// TwinCAT 3 PLC project ElevatorControl
// ProgramVersion: 3.1.4024.0
// libraries:
//   Tc2_Standard, * (Beckhoff Automation GmbH)
//   Tc2_System, * (Beckhoff Automation GmbH)
//   Tc2_Utilities, * (Beckhoff Automation GmbH)
//   Tc3_Module, * (Beckhoff Automation GmbH)
// project tree:
//   DUTs/ AT_AlarmLog.TcDUT (not stored), AT_FloorCalls.TcDUT (not stored), E_AlarmSeverity.TcDUT (not stored), E_Direction.TcDUT (not stored), E_ElevatorState.TcDUT, E_TrafficMode.TcDUT (not stored), ST_AlarmEvent.TcDUT (not stored), ST_ElevatorStatus.TcDUT, ST_FloorCall.TcDUT, ST_PerformanceMetrics.TcDUT (not stored)
//   GVLs/ GVL_HMI.TcGVL, GVL_IO.TcGVL (not stored), GVL_Parameters.TcGVL (not stored)
//   / PlcTask.TcTTO
//   POUs/ FB_Elevator.TcPOU (not stored), FB_Safety.TcPOU, MAIN.TcPOU, FB_Dispatcher.TcPOU, PRG_Test_Elevator.TcPOU
// real-time tasks:
//   TASK PlcTask: cycle T#10ms, priority 20, ADS port 350
//   TASK PlcTask1: cycle T#10ms, priority 21, ADS port 351

CONFIGURATION ElevatorControl
    RESOURCE PLC ON TwinCAT3
        TASK PlcTask(INTERVAL := T#10ms, PRIORITY := 20);
        PROGRAM MAIN WITH PlcTask : MAIN;
    END_RESOURCE
END_CONFIGURATION

// ---- DUTs/E_ElevatorState.TcDUT
{attribute 'qualified_only'}
{attribute 'strict'}
TYPE E_ElevatorState :
(
	eIdle           := 0,   // Waiting for calls, doors closed
    eMovingUp       := 1,   // Traveling upward
    eMovingDown     := 2,   // Traveling downward
    eDoorsOpening   := 3,   // Door opening animation
    eDoorsOpen      := 4,   // Doors fully open, waiting for passengers
    eDoorsClosing   := 5,   // Door closing animation
    eEmergencyStop  := 6,   // Emergency stop button pressed
    eFireMode       := 7,   // Fire alarm — returning to ground
    eOverload       := 8,   // Too much weight detected
    eMaintenance    := 9    // Service mode (future feature)
);
END_TYPE

// ---- DUTs/ST_ElevatorStatus.TcDUT
TYPE ST_ElevatorStatus :
STRUCT
    iElevatorID     : INT;              // 1 = E1, 2 = E2
    iCurrentFloor   : INT;              // Which floor it's at (0-10)
    fPosition       : REAL;             // Smooth position 0.0-10.0 for animation
    eState          : E_ElevatorState;  // What it's doing right now
    eDirection      : E_Direction;      // Which way it's going
    bDoorsOpen      : BOOL;             // TRUE = doors are open
    fDoorOpenPercent: REAL;             // 0.0-100.0 for door animation width
    iNextTarget     : INT;              // Next floor it's going to (-1 = none)
    iQueueLength    : INT;              // How many calls pending
    bOverload       : BOOL;             // TRUE = too heavy
    bDoorObstruction: BOOL;             // TRUE = something blocking door
    fTravelDistance : REAL;             // Total meters traveled (maintenance metric)
    iTripCount      : DINT;             // Total completed trips
    tLastMaintenance: TIME;             // Time since last service
END_STRUCT
END_TYPE

// ---- DUTs/ST_FloorCall.TcDUT
TYPE ST_FloorCall :
STRUCT
    iFloor          : INT;          // Which floor (0 = Ground, 1-10)
    eDirection      : E_Direction;  // For hall buttons: Up or Down
    bIsCarCall      : BOOL;         // TRUE = pressed inside elevator, FALSE = hallway
    tTimestamp      : TIME;         // When the button was pressed
    iAssignedTo     : INT;          // 0 = not assigned yet, 1 = E1, 2 = E2
    bIsActive       : BOOL;         // TRUE = still waiting, FALSE = completed
    tWaitTime       : TIME;         // How long the person has been waiting
END_STRUCT
END_TYPE

// ---- GVLs/GVL_HMI.TcGVL
{attribute 'qualified_only'}
// ============================================
// GVL_HMI — Variables Exposed to HMI
// ============================================

VAR_GLOBAL
    // Elevator status — what the HMI displays
    g_stE1Status        : ST_ElevatorStatus;    // Everything about E1
    g_stE2Status        : ST_ElevatorStatus;    // Everything about E2
    
    // System metrics
    g_stMetrics         : ST_PerformanceMetrics;
    
    // Alarm history
    g_astAlarmLog       : AT_AlarmLog;
    g_iAlarmCount       : INT := 0;
    
    // Call queue display
    g_astCallQueue      : AT_FloorCalls;
    g_iQueueCount       : INT := 0;
    
    // System status text
    g_bSystemReady      		: BOOL := FALSE;
    g_sSystemStatus     		: STRING(40) := 'Initializing';
    g_bAlarmActive      		: BOOL := FALSE;
    g_sAlarmMessage     		: STRING(120) := '';
	g_bHMI_ResetAlarmEnabled 	: BOOL := FALSE;
    
    // ------------------------------------------------------------------------
    // HMI TO PLC — Commands from operator
    // ------------------------------------------------------------------------
    g_bHMI_EmergencyStop    : BOOL := FALSE;    // Pressed = stop everything
    g_bHMI_ResetEmergency   : BOOL := FALSE;    // Pressed = clear emergency
    g_bHMI_FireMode         : BOOL := FALSE;    // Pressed = activate fire mode
    g_bHMI_ResetFireMode    : BOOL := FALSE;    // Pressed = clear fire mode
    g_eHMI_TrafficMode      : E_TrafficMode := E_TrafficMode.eOffPeak;
    g_bHMI_ClearAllCalls    : BOOL := FALSE;    // Pressed = empty all queues
	g_bHMI_ResetAlarm 		: BOOL := FALSE;	// Pressed = reset active alarms
    
    // ------------------------------------------------------------------------
    // HMI TO PLC — Floor calls from HMI buttons
    // ------------------------------------------------------------------------
    // Hall calls
    g_bHMI_Call_G_Up        : BOOL := FALSE;
    g_bHMI_Call_1_Up        : BOOL := FALSE;
    g_bHMI_Call_1_Down      : BOOL := FALSE;
    g_bHMI_Call_2_Up        : BOOL := FALSE;
    g_bHMI_Call_2_Down      : BOOL := FALSE;
    g_bHMI_Call_3_Up        : BOOL := FALSE;
    g_bHMI_Call_3_Down      : BOOL := FALSE;
    g_bHMI_Call_4_Up        : BOOL := FALSE;
    g_bHMI_Call_4_Down      : BOOL := FALSE;
    g_bHMI_Call_5_Up        : BOOL := FALSE;
    g_bHMI_Call_5_Down      : BOOL := FALSE;
    g_bHMI_Call_6_Up        : BOOL := FALSE;
    g_bHMI_Call_6_Down      : BOOL := FALSE;
    g_bHMI_Call_7_Up        : BOOL := FALSE;
    g_bHMI_Call_7_Down      : BOOL := FALSE;
    g_bHMI_Call_8_Up        : BOOL := FALSE;
    g_bHMI_Call_8_Down      : BOOL := FALSE;
    g_bHMI_Call_9_Up        : BOOL := FALSE;
    g_bHMI_Call_9_Down      : BOOL := FALSE;
    g_bHMI_Call_10_Down     : BOOL := FALSE;
    
    // Car calls — Elevator 1
    g_bHMI_E1_Car_G         : BOOL := FALSE;
    g_bHMI_E1_Car_1         : BOOL := FALSE;
    g_bHMI_E1_Car_2         : BOOL := FALSE;
    g_bHMI_E1_Car_3         : BOOL := FALSE;
    g_bHMI_E1_Car_4         : BOOL := FALSE;
    g_bHMI_E1_Car_5         : BOOL := FALSE;
    g_bHMI_E1_Car_6         : BOOL := FALSE;
    g_bHMI_E1_Car_7         : BOOL := FALSE;
    g_bHMI_E1_Car_8         : BOOL := FALSE;
    g_bHMI_E1_Car_9         : BOOL := FALSE;
    g_bHMI_E1_Car_10        : BOOL := FALSE;
    
    // Car calls — Elevator 2
    g_bHMI_E2_Car_G         : BOOL := FALSE;
    g_bHMI_E2_Car_1         : BOOL := FALSE;
    g_bHMI_E2_Car_2         : BOOL := FALSE;
    g_bHMI_E2_Car_3         : BOOL := FALSE;
    g_bHMI_E2_Car_4         : BOOL := FALSE;
    g_bHMI_E2_Car_5         : BOOL := FALSE;
    g_bHMI_E2_Car_6         : BOOL := FALSE;
    g_bHMI_E2_Car_7         : BOOL := FALSE;
    g_bHMI_E2_Car_8         : BOOL := FALSE;
    g_bHMI_E2_Car_9         : BOOL := FALSE;
    g_bHMI_E2_Car_10        : BOOL := FALSE;
    
END_VAR

// ---- POUs/MAIN.TcPOU
PROGRAM MAIN

// ============================================================================
// ELEVATOR INSTANCES
// ============================================================================
VAR
    E1              : FB_Elevator;
    E2              : FB_Elevator;
	
	 prgTestElevator : PRG_Test_Elevator;

END_VAR

// ============================================================================
// GROUP CONTROL
// ============================================================================
VAR
    Dispatcher      : FB_Dispatcher;
END_VAR

// ============================================================================
// SAFETY SYSTEM
// ============================================================================
VAR
    Safety          : FB_Safety;
END_VAR

// ============================================================================
// SIMULATION INPUTS (Delete these when connecting real hardware)
// ============================================================================
VAR
    // Hall call simulation
    bSimHall_G_Up       : BOOL := FALSE;
    bSimHall_1_Up       : BOOL := FALSE;
    bSimHall_1_Down     : BOOL := FALSE;
    bSimHall_2_Up       : BOOL := FALSE;
    bSimHall_2_Down     : BOOL := FALSE;
    bSimHall_3_Up       : BOOL := FALSE;
    bSimHall_3_Down     : BOOL := FALSE;
    bSimHall_4_Up       : BOOL := FALSE;
    bSimHall_4_Down     : BOOL := FALSE;
    bSimHall_5_Up       : BOOL := FALSE;
    bSimHall_5_Down     : BOOL := FALSE;
    bSimHall_6_Up       : BOOL := FALSE;
    bSimHall_6_Down     : BOOL := FALSE;
    bSimHall_7_Up       : BOOL := FALSE;
    bSimHall_7_Down     : BOOL := FALSE;
    bSimHall_8_Up       : BOOL := FALSE;
    bSimHall_8_Down     : BOOL := FALSE;
    bSimHall_9_Up       : BOOL := FALSE;
    bSimHall_9_Down     : BOOL := FALSE;
    bSimHall_10_Down    : BOOL := FALSE;
    
    // Car call simulation — E1
    bSimE1_Car_G        : BOOL := FALSE;
    bSimE1_Car_1        : BOOL := FALSE;
    bSimE1_Car_2        : BOOL := FALSE;
    bSimE1_Car_3        : BOOL := FALSE;
    bSimE1_Car_4        : BOOL := FALSE;
    bSimE1_Car_5        : BOOL := FALSE;
    bSimE1_Car_6        : BOOL := FALSE;
    bSimE1_Car_7        : BOOL := FALSE;
    bSimE1_Car_8        : BOOL := FALSE;
    bSimE1_Car_9        : BOOL := FALSE;
    bSimE1_Car_10       : BOOL := FALSE;
    
    // Car call simulation — E2
    bSimE2_Car_G        : BOOL := FALSE;
    bSimE2_Car_1        : BOOL := FALSE;
    bSimE2_Car_2        : BOOL := FALSE;
    bSimE2_Car_3        : BOOL := FALSE;
    bSimE2_Car_4        : BOOL := FALSE;
    bSimE2_Car_5        : BOOL := FALSE;
    bSimE2_Car_6        : BOOL := FALSE;
    bSimE2_Car_7        : BOOL := FALSE;
    bSimE2_Car_8        : BOOL := FALSE;
    bSimE2_Car_9        : BOOL := FALSE;
    bSimE2_Car_10       : BOOL := FALSE;
    
    // Safety simulation
    bSimE1_DoorSensor   : BOOL := FALSE;
    bSimE1_WeightSensor : BOOL := FALSE;
    bSimE1_EmergencyBtn : BOOL := FALSE;
    bSimE2_DoorSensor   : BOOL := FALSE;
    bSimE2_WeightSensor : BOOL := FALSE;
    bSimE2_EmergencyBtn : BOOL := FALSE;
    bSimFireAlarm       : BOOL := FALSE;
    bSimPowerFault      : BOOL := FALSE;
    
    // HMI command simulation
    bSimHMI_EmergencyStop   : BOOL := FALSE;
    bSimHMI_ResetEmergency  : BOOL := FALSE;
    bSimHMI_FireMode        : BOOL := FALSE;
    bSimHMI_ResetFireMode   : BOOL := FALSE;
    bSimHMI_ClearAllCalls   : BOOL := FALSE;
END_VAR

// ============================================================================
// INTERNAL STATE TRACKING
// ============================================================================
VAR
    _bInitialized       : BOOL := FALSE;
    _bPrevClearCalls    : BOOL := FALSE;
	 bSystemEnable 		: BOOL := TRUE;
END_VAR

prgTestElevator();

// ======================================================================
// ONE-TIME INITIALIZATION
// ======================================================================
IF NOT _bInitialized THEN
    
    // Connect dispatcher references to elevator instances
    Dispatcher.refE1 REF= E1;
    Dispatcher.refE2 REF= E2;
    
    // Connect safety references to elevator instances
    Safety.refE1 REF= E1;
    Safety.refE2 REF= E2;
    
    _bInitialized := TRUE;
    
END_IF;

// ======================================================================
// SIMULATION: COPY SIM INPUTS TO PHYSICAL I/O ADDRESSES
// ======================================================================
// DELETE THIS ENTIRE SECTION WHEN CONNECTING REAL HARDWARE
// ----------------------------------------------------------------------

// Hall calls
GVL_IO.diHall_G_Up         := bSimHall_G_Up;
GVL_IO.diHall_1_Up         := bSimHall_1_Up;
GVL_IO.diHall_1_Down       := bSimHall_1_Down;
GVL_IO.diHall_2_Up         := bSimHall_2_Up;
GVL_IO.diHall_2_Down       := bSimHall_2_Down;
GVL_IO.diHall_3_Up         := bSimHall_3_Up;
GVL_IO.diHall_3_Down       := bSimHall_3_Down;
GVL_IO.diHall_4_Up         := bSimHall_4_Up;
GVL_IO.diHall_4_Down       := bSimHall_4_Down;
GVL_IO.diHall_5_Up         := bSimHall_5_Up;
GVL_IO.diHall_5_Down       := bSimHall_5_Down;
GVL_IO.diHall_6_Up         := bSimHall_6_Up;
GVL_IO.diHall_6_Down       := bSimHall_6_Down;
GVL_IO.diHall_7_Up         := bSimHall_7_Up;
GVL_IO.diHall_7_Down       := bSimHall_7_Down;
GVL_IO.diHall_8_Up         := bSimHall_8_Up;
GVL_IO.diHall_8_Down       := bSimHall_8_Down;
GVL_IO.diHall_9_Up         := bSimHall_9_Up;
GVL_IO.diHall_9_Down       := bSimHall_9_Down;
GVL_IO.diHall_10_Down      := bSimHall_10_Down;

// Car calls E1
GVL_IO.diE1_Car_G          := bSimE1_Car_G;
GVL_IO.diE1_Car_1          := bSimE1_Car_1;
GVL_IO.diE1_Car_2          := bSimE1_Car_2;
GVL_IO.diE1_Car_3          := bSimE1_Car_3;
GVL_IO.diE1_Car_4          := bSimE1_Car_4;
GVL_IO.diE1_Car_5          := bSimE1_Car_5;
GVL_IO.diE1_Car_6          := bSimE1_Car_6;
GVL_IO.diE1_Car_7          := bSimE1_Car_7;
GVL_IO.diE1_Car_8          := bSimE1_Car_8;
GVL_IO.diE1_Car_9          := bSimE1_Car_9;
GVL_IO.diE1_Car_10         := bSimE1_Car_10;

// Car calls E2
GVL_IO.diE2_Car_G          := bSimE2_Car_G;
GVL_IO.diE2_Car_1          := bSimE2_Car_1;
GVL_IO.diE2_Car_2          := bSimE2_Car_2;
GVL_IO.diE2_Car_3          := bSimE2_Car_3;
GVL_IO.diE2_Car_4          := bSimE2_Car_4;
GVL_IO.diE2_Car_5          := bSimE2_Car_5;
GVL_IO.diE2_Car_6          := bSimE2_Car_6;
GVL_IO.diE2_Car_7          := bSimE2_Car_7;
GVL_IO.diE2_Car_8          := bSimE2_Car_8;
GVL_IO.diE2_Car_9          := bSimE2_Car_9;
GVL_IO.diE2_Car_10         := bSimE2_Car_10;

// Safety sensors
GVL_IO.diE1_DoorSensor     := bSimE1_DoorSensor;
GVL_IO.diE1_WeightSensor   := bSimE1_WeightSensor;
GVL_IO.diE1_EmergencyBtn   := bSimE1_EmergencyBtn;
GVL_IO.diE2_DoorSensor     := bSimE2_DoorSensor;
GVL_IO.diE2_WeightSensor   := bSimE2_WeightSensor;
GVL_IO.diE2_EmergencyBtn   := bSimE2_EmergencyBtn;
GVL_IO.diFireAlarm         := bSimFireAlarm;
GVL_IO.diPowerFault        := bSimPowerFault;

// HMI commands
GVL_HMI.g_bHMI_EmergencyStop    := bSimHMI_EmergencyStop;
GVL_HMI.g_bHMI_ResetEmergency   := bSimHMI_ResetEmergency;
GVL_HMI.g_bHMI_FireMode         := bSimHMI_FireMode;
GVL_HMI.g_bHMI_ResetFireMode    := bSimHMI_ResetFireMode;
GVL_HMI.g_bHMI_ClearAllCalls    := bSimHMI_ClearAllCalls;

// ======================================================================
// MAP PHYSICAL I/O TO ELEVATOR INPUTS
// ======================================================================

// Elevator 1 inputs
E1.bEnable          := bSystemEnable AND Safety.bE1Enable;
E1.bEmergencyStop   := GVL_IO.diE1_EmergencyBtn OR GVL_HMI.g_bHMI_EmergencyStop;
E1.bFireMode        := GVL_IO.diFireAlarm OR GVL_HMI.g_bHMI_FireMode;
E1.bDoorObstruction := GVL_IO.diE1_DoorSensor;
E1.bOverload        := GVL_IO.diE1_WeightSensor;

// Elevator 2 inputs
E2.bEnable          := bSystemEnable AND Safety.bE2Enable;
E2.bEmergencyStop   := GVL_IO.diE2_EmergencyBtn OR GVL_HMI.g_bHMI_EmergencyStop;
E2.bFireMode        := GVL_IO.diFireAlarm OR GVL_HMI.g_bHMI_FireMode;
E2.bDoorObstruction := GVL_IO.diE2_DoorSensor;
E2.bOverload        := GVL_IO.diE2_WeightSensor;

// ======================================================================
// MAP PHYSICAL I/O TO SAFETY INPUTS
// ======================================================================
Safety.bE1DoorSensor    := GVL_IO.diE1_DoorSensor;
Safety.bE2DoorSensor    := GVL_IO.diE2_DoorSensor;
Safety.bE1WeightSensor  := GVL_IO.diE1_WeightSensor;
Safety.bE2WeightSensor  := GVL_IO.diE2_WeightSensor;
Safety.bE1EmergencyBtn  := GVL_IO.diE1_EmergencyBtn;
Safety.bE2EmergencyBtn  := GVL_IO.diE2_EmergencyBtn;
Safety.bFireAlarm       := GVL_IO.diFireAlarm;
Safety.bPowerFault      := GVL_IO.diPowerFault;

// ======================================================================
// PROCESS HALL CALLS → DISPATCHER
// ======================================================================
IF GVL_IO.diHall_G_Up      THEN Dispatcher.AddCall(0, E_Direction.eUp, FALSE, 0); END_IF;
IF GVL_IO.diHall_1_Up      THEN Dispatcher.AddCall(1, E_Direction.eUp, FALSE, 0); END_IF;
IF GVL_IO.diHall_1_Down    THEN Dispatcher.AddCall(1, E_Direction.eDown, FALSE, 0); END_IF;
IF GVL_IO.diHall_2_Up      THEN Dispatcher.AddCall(2, E_Direction.eUp, FALSE, 0); END_IF;
IF GVL_IO.diHall_2_Down    THEN Dispatcher.AddCall(2, E_Direction.eDown, FALSE, 0); END_IF;
IF GVL_IO.diHall_3_Up      THEN Dispatcher.AddCall(3, E_Direction.eUp, FALSE, 0); END_IF;
IF GVL_IO.diHall_3_Down    THEN Dispatcher.AddCall(3, E_Direction.eDown, FALSE, 0); END_IF;
IF GVL_IO.diHall_4_Up      THEN Dispatcher.AddCall(4, E_Direction.eUp, FALSE, 0); END_IF;
IF GVL_IO.diHall_4_Down    THEN Dispatcher.AddCall(4, E_Direction.eDown, FALSE, 0); END_IF;
IF GVL_IO.diHall_5_Up      THEN Dispatcher.AddCall(5, E_Direction.eUp, FALSE, 0); END_IF;
IF GVL_IO.diHall_5_Down    THEN Dispatcher.AddCall(5, E_Direction.eDown, FALSE, 0); END_IF;
IF GVL_IO.diHall_6_Up      THEN Dispatcher.AddCall(6, E_Direction.eUp, FALSE, 0); END_IF;
IF GVL_IO.diHall_6_Down    THEN Dispatcher.AddCall(6, E_Direction.eDown, FALSE, 0); END_IF;
IF GVL_IO.diHall_7_Up      THEN Dispatcher.AddCall(7, E_Direction.eUp, FALSE, 0); END_IF;
IF GVL_IO.diHall_7_Down    THEN Dispatcher.AddCall(7, E_Direction.eDown, FALSE, 0); END_IF;
IF GVL_IO.diHall_8_Up      THEN Dispatcher.AddCall(8, E_Direction.eUp, FALSE, 0); END_IF;
IF GVL_IO.diHall_8_Down    THEN Dispatcher.AddCall(8, E_Direction.eDown, FALSE, 0); END_IF;
IF GVL_IO.diHall_9_Up      THEN Dispatcher.AddCall(9, E_Direction.eUp, FALSE, 0); END_IF;
IF GVL_IO.diHall_9_Down    THEN Dispatcher.AddCall(9, E_Direction.eDown, FALSE, 0); END_IF;
IF GVL_IO.diHall_10_Down   THEN Dispatcher.AddCall(10, E_Direction.eDown, FALSE, 0); END_IF;

// ======================================================================
// PROCESS CAR CALLS → DIRECT TO ELEVATOR
// ======================================================================
IF GVL_IO.diE1_Car_G   THEN E1.CallFloor(0); END_IF;
IF GVL_IO.diE1_Car_1   THEN E1.CallFloor(1); END_IF;
IF GVL_IO.diE1_Car_2   THEN E1.CallFloor(2); END_IF;
IF GVL_IO.diE1_Car_3   THEN E1.CallFloor(3); END_IF;
IF GVL_IO.diE1_Car_4   THEN E1.CallFloor(4); END_IF;
IF GVL_IO.diE1_Car_5   THEN E1.CallFloor(5); END_IF;
IF GVL_IO.diE1_Car_6   THEN E1.CallFloor(6); END_IF;
IF GVL_IO.diE1_Car_7   THEN E1.CallFloor(7); END_IF;
IF GVL_IO.diE1_Car_8   THEN E1.CallFloor(8); END_IF;
IF GVL_IO.diE1_Car_9   THEN E1.CallFloor(9); END_IF;
IF GVL_IO.diE1_Car_10  THEN E1.CallFloor(10); END_IF;

IF GVL_IO.diE2_Car_G   THEN E2.CallFloor(0); END_IF;
IF GVL_IO.diE2_Car_1   THEN E2.CallFloor(1); END_IF;
IF GVL_IO.diE2_Car_2   THEN E2.CallFloor(2); END_IF;
IF GVL_IO.diE2_Car_3   THEN E2.CallFloor(3); END_IF;
IF GVL_IO.diE2_Car_4   THEN E2.CallFloor(4); END_IF;
IF GVL_IO.diE2_Car_5   THEN E2.CallFloor(5); END_IF;
IF GVL_IO.diE2_Car_6   THEN E2.CallFloor(6); END_IF;
IF GVL_IO.diE2_Car_7   THEN E2.CallFloor(7); END_IF;
IF GVL_IO.diE2_Car_8   THEN E2.CallFloor(8); END_IF;
IF GVL_IO.diE2_Car_9   THEN E2.CallFloor(9); END_IF;
IF GVL_IO.diE2_Car_10  THEN E2.CallFloor(10); END_IF;

// ======================================================================
// HMI CAR CALLS
// ======================================================================
IF GVL_HMI.g_bHMI_E1_Car_G THEN E1.CallFloor(0); GVL_HMI.g_bHMI_E1_Car_G := FALSE; END_IF;
IF GVL_HMI.g_bHMI_E1_Car_1 THEN E1.CallFloor(1); GVL_HMI.g_bHMI_E1_Car_1 := FALSE; END_IF;
IF GVL_HMI.g_bHMI_E1_Car_2 THEN E1.CallFloor(2); GVL_HMI.g_bHMI_E1_Car_2 := FALSE; END_IF;
IF GVL_HMI.g_bHMI_E1_Car_3 THEN E1.CallFloor(3); GVL_HMI.g_bHMI_E1_Car_3 := FALSE; END_IF;
IF GVL_HMI.g_bHMI_E1_Car_4 THEN E1.CallFloor(4); GVL_HMI.g_bHMI_E1_Car_4 := FALSE; END_IF;
IF GVL_HMI.g_bHMI_E1_Car_5 THEN E1.CallFloor(5); GVL_HMI.g_bHMI_E1_Car_5 := FALSE; END_IF;
IF GVL_HMI.g_bHMI_E1_Car_6 THEN E1.CallFloor(6); GVL_HMI.g_bHMI_E1_Car_6 := FALSE; END_IF;
IF GVL_HMI.g_bHMI_E1_Car_7 THEN E1.CallFloor(7); GVL_HMI.g_bHMI_E1_Car_7 := FALSE; END_IF;
IF GVL_HMI.g_bHMI_E1_Car_8 THEN E1.CallFloor(8); GVL_HMI.g_bHMI_E1_Car_8 := FALSE; END_IF;
IF GVL_HMI.g_bHMI_E1_Car_9 THEN E1.CallFloor(9); GVL_HMI.g_bHMI_E1_Car_9 := FALSE; END_IF;
IF GVL_HMI.g_bHMI_E1_Car_10 THEN E1.CallFloor(10); GVL_HMI.g_bHMI_E1_Car_10 := FALSE; END_IF;

IF GVL_HMI.g_bHMI_E2_Car_G THEN E2.CallFloor(0); GVL_HMI.g_bHMI_E2_Car_G := FALSE; END_IF;
IF GVL_HMI.g_bHMI_E2_Car_1 THEN E2.CallFloor(1); GVL_HMI.g_bHMI_E2_Car_1 := FALSE; END_IF;
IF GVL_HMI.g_bHMI_E2_Car_2 THEN E2.CallFloor(2); GVL_HMI.g_bHMI_E2_Car_2 := FALSE; END_IF;
IF GVL_HMI.g_bHMI_E2_Car_3 THEN E2.CallFloor(3); GVL_HMI.g_bHMI_E2_Car_3 := FALSE; END_IF;
IF GVL_HMI.g_bHMI_E2_Car_4 THEN E2.CallFloor(4); GVL_HMI.g_bHMI_E2_Car_4 := FALSE; END_IF;
IF GVL_HMI.g_bHMI_E2_Car_5 THEN E2.CallFloor(5); GVL_HMI.g_bHMI_E2_Car_5 := FALSE; END_IF;
IF GVL_HMI.g_bHMI_E2_Car_6 THEN E2.CallFloor(6); GVL_HMI.g_bHMI_E2_Car_6 := FALSE; END_IF;
IF GVL_HMI.g_bHMI_E2_Car_7 THEN E2.CallFloor(7); GVL_HMI.g_bHMI_E2_Car_7 := FALSE; END_IF;
IF GVL_HMI.g_bHMI_E2_Car_8 THEN E2.CallFloor(8); GVL_HMI.g_bHMI_E2_Car_8 := FALSE; END_IF;
IF GVL_HMI.g_bHMI_E2_Car_9 THEN E2.CallFloor(9); GVL_HMI.g_bHMI_E2_Car_9 := FALSE; END_IF;
IF GVL_HMI.g_bHMI_E2_Car_10 THEN E2.CallFloor(10); GVL_HMI.g_bHMI_E2_Car_10 := FALSE; END_IF;

// ======================================================================
// HMI HALL CALLS
// ======================================================================
IF GVL_HMI.g_bHMI_Call_G_Up THEN Dispatcher.AddCall(0, E_Direction.eUp, FALSE, 0); GVL_HMI.g_bHMI_Call_G_Up := FALSE; END_IF;
IF GVL_HMI.g_bHMI_Call_1_Up THEN Dispatcher.AddCall(1, E_Direction.eUp, FALSE, 0); GVL_HMI.g_bHMI_Call_1_Up := FALSE; END_IF;
IF GVL_HMI.g_bHMI_Call_1_Down THEN Dispatcher.AddCall(1, E_Direction.eDown, FALSE, 0); GVL_HMI.g_bHMI_Call_1_Down := FALSE; END_IF;
IF GVL_HMI.g_bHMI_Call_2_Up THEN Dispatcher.AddCall(2, E_Direction.eUp, FALSE, 0); GVL_HMI.g_bHMI_Call_2_Up := FALSE; END_IF;
IF GVL_HMI.g_bHMI_Call_2_Down THEN Dispatcher.AddCall(2, E_Direction.eDown, FALSE, 0); GVL_HMI.g_bHMI_Call_2_Down := FALSE; END_IF;
IF GVL_HMI.g_bHMI_Call_3_Up THEN Dispatcher.AddCall(3, E_Direction.eUp, FALSE, 0); GVL_HMI.g_bHMI_Call_3_Up := FALSE; END_IF;
IF GVL_HMI.g_bHMI_Call_3_Down THEN Dispatcher.AddCall(3, E_Direction.eDown, FALSE, 0); GVL_HMI.g_bHMI_Call_3_Down := FALSE; END_IF;
IF GVL_HMI.g_bHMI_Call_4_Up THEN Dispatcher.AddCall(4, E_Direction.eUp, FALSE, 0); GVL_HMI.g_bHMI_Call_4_Up := FALSE; END_IF;
IF GVL_HMI.g_bHMI_Call_4_Down THEN Dispatcher.AddCall(4, E_Direction.eDown, FALSE, 0); GVL_HMI.g_bHMI_Call_4_Down := FALSE; END_IF;
IF GVL_HMI.g_bHMI_Call_5_Up THEN Dispatcher.AddCall(5, E_Direction.eUp, FALSE, 0); GVL_HMI.g_bHMI_Call_5_Up := FALSE; END_IF;
IF GVL_HMI.g_bHMI_Call_5_Down THEN Dispatcher.AddCall(5, E_Direction.eDown, FALSE, 0); GVL_HMI.g_bHMI_Call_5_Down := FALSE; END_IF;
IF GVL_HMI.g_bHMI_Call_6_Up THEN Dispatcher.AddCall(6, E_Direction.eUp, FALSE, 0); GVL_HMI.g_bHMI_Call_6_Up := FALSE; END_IF;
IF GVL_HMI.g_bHMI_Call_6_Down THEN Dispatcher.AddCall(6, E_Direction.eDown, FALSE, 0); GVL_HMI.g_bHMI_Call_6_Down := FALSE; END_IF;
IF GVL_HMI.g_bHMI_Call_7_Up THEN Dispatcher.AddCall(7, E_Direction.eUp, FALSE, 0); GVL_HMI.g_bHMI_Call_7_Up := FALSE; END_IF;
IF GVL_HMI.g_bHMI_Call_7_Down THEN Dispatcher.AddCall(7, E_Direction.eDown, FALSE, 0); GVL_HMI.g_bHMI_Call_7_Down := FALSE; END_IF;
IF GVL_HMI.g_bHMI_Call_8_Up THEN Dispatcher.AddCall(8, E_Direction.eUp, FALSE, 0); GVL_HMI.g_bHMI_Call_8_Up := FALSE; END_IF;
IF GVL_HMI.g_bHMI_Call_8_Down THEN Dispatcher.AddCall(8, E_Direction.eDown, FALSE, 0); GVL_HMI.g_bHMI_Call_8_Down := FALSE; END_IF;
IF GVL_HMI.g_bHMI_Call_9_Up THEN Dispatcher.AddCall(9, E_Direction.eUp, FALSE, 0); GVL_HMI.g_bHMI_Call_9_Up := FALSE; END_IF;
IF GVL_HMI.g_bHMI_Call_9_Down THEN Dispatcher.AddCall(9, E_Direction.eDown, FALSE, 0); GVL_HMI.g_bHMI_Call_9_Down := FALSE; END_IF;
IF GVL_HMI.g_bHMI_Call_10_Down THEN Dispatcher.AddCall(10, E_Direction.eDown, FALSE, 0); GVL_HMI.g_bHMI_Call_10_Down := FALSE; END_IF;

// ======================================================================
// RESET ACTIVE ALARM (HMI command)
// ======================================================================
IF GVL_HMI.g_bHMI_ResetAlarm THEN
    IF Safety.ResetSystemAlarm() THEN
        GVL_HMI.g_bHMI_ResetAlarm := FALSE;
    END_IF
END_IF;

// ======================================================================
// CLEAR ALL CALLS
// ======================================================================
IF GVL_HMI.g_bHMI_ClearAllCalls AND NOT _bPrevClearCalls THEN
    Dispatcher.ClearAllCalls();
    E1.ClearCall(0); E1.ClearCall(1); E1.ClearCall(2); E1.ClearCall(3);
    E1.ClearCall(4); E1.ClearCall(5); E1.ClearCall(6); E1.ClearCall(7);
    E1.ClearCall(8); E1.ClearCall(9); E1.ClearCall(10);
    E2.ClearCall(0); E2.ClearCall(1); E2.ClearCall(2); E2.ClearCall(3);
    E2.ClearCall(4); E2.ClearCall(5); E2.ClearCall(6); E2.ClearCall(7);
    E2.ClearCall(8); E2.ClearCall(9); E2.ClearCall(10);
END_IF;

_bPrevClearCalls := GVL_HMI.g_bHMI_ClearAllCalls;

// ======================================================================
// CYCLIC EXECUTION — CALL ALL FBs EVERY SCAN
// ======================================================================

// Run elevators
E1();
E2();

// Run dispatcher
Dispatcher.ProcessQueue();
Dispatcher.eTrafficMode := GVL_HMI.g_eHMI_TrafficMode;

// Run safety
Safety();

// ======================================================================
// UPDATE HMI OUTPUT DATA
// ======================================================================
GVL_HMI.g_stE1Status := E1.GetStatus();
GVL_HMI.g_stE2Status := E2.GetStatus();
GVL_HMI.g_stMetrics := Dispatcher.stMetrics;
GVL_HMI.g_astAlarmLog := Safety.GetAlarmLog();
GVL_HMI.g_bSystemReady := E1.bIsReady OR E2.bIsReady;
GVL_HMI.g_bAlarmActive := Safety.bSystemAlarm;
GVL_HMI.g_bHMI_ResetAlarmEnabled := Safety.bSystemAlarm;

IF Safety.bSystemAlarm THEN
    GVL_HMI.g_sAlarmMessage := Safety.sAlarmMessage;
ELSE
    GVL_HMI.g_sAlarmMessage := '';
END_IF;

// System status text
IF E1.eState = E_ElevatorState.eEmergencyStop OR 
   E2.eState = E_ElevatorState.eEmergencyStop THEN
    GVL_HMI.g_sSystemStatus := 'EMERGENCY STOP';
ELSIF E1.eState = E_ElevatorState.eFireMode OR 	
      E2.eState = E_ElevatorState.eFireMode THEN
    GVL_HMI.g_sSystemStatus := 'FIRE MODE ACTIVE';
ELSIF NOT bSystemEnable THEN
    GVL_HMI.g_sSystemStatus := 'SYSTEM DISABLED';
ELSE
    GVL_HMI.g_sSystemStatus := 'NORMAL OPERATION';
END_IF;

END_PROGRAM

// ---- POUs/PRG_Test_Elevator.TcPOU
FUNCTION_BLOCK PRG_Test_Elevator
VAR
    // Instance under test
    fbElev  : FB_Elevator;
    
    // Test control
    nStep       : INT := 0;
    bDone       : BOOL := FALSE;
    bPassed     : BOOL := FALSE;
    
    // Step timer
    tonWait     : TON;
    
    // Call tracking
    bCalledFloor3   : BOOL := FALSE;
    bCalledFloor1   : BOOL := FALSE;
END_VAR

// ============================================
// ELEVATOR UNIT TEST — Automatic Sequence
// ============================================

IF bDone THEN
    RETURN; // Test finished, keep results visible
END_IF;

CASE nStep OF

// --------------------------------------------
// STEP 0: Verify initial state
// --------------------------------------------
0:
    IF fbElev.eState = E_ElevatorState.eIdle AND 
       fbElev.iCurrentFloor = 0 AND
       fbElev.fDoorOpenPercent = 0.0 THEN
        nStep := 1;
    END_IF;

// --------------------------------------------
// STEP 1: Call elevator to floor 3
// --------------------------------------------
1:
    fbElev.bEnable := TRUE;
    IF NOT bCalledFloor3 THEN
        fbElev.CallFloor(3);
        bCalledFloor3 := TRUE;
    END_IF;
    
    // Should start moving up
    IF fbElev.eState = E_ElevatorState.eMovingUp THEN
        nStep := 2;
    END_IF;

// --------------------------------------------
// STEP 2: Wait until doors open at floor 3
// --------------------------------------------
2:
    IF fbElev.iCurrentFloor = 3 AND 
       fbElev.eState = E_ElevatorState.eDoorsOpen AND
       fbElev.fDoorOpenPercent >= 99.0 THEN
        nStep := 3;
        tonWait(IN := FALSE); // Reset timer
    END_IF;

// --------------------------------------------
// STEP 3: Wait for doors to close, return to idle
// --------------------------------------------
3:
    tonWait(IN := TRUE, PT := T#5S); // Give time for full cycle
    
    IF fbElev.eState = E_ElevatorState.eIdle AND tonWait.Q THEN
        nStep := 4;
        bCalledFloor1 := FALSE;
    END_IF;

// --------------------------------------------
// STEP 4: Call floor 1 (going down)
// --------------------------------------------
4:
    IF NOT bCalledFloor1 THEN
        fbElev.CallFloor(1);
        bCalledFloor1 := TRUE;
    END_IF;
    
    IF fbElev.eState = E_ElevatorState.eMovingDown THEN
        nStep := 5;
    END_IF;

// --------------------------------------------
// STEP 5: Arrive at floor 1, verify complete
// --------------------------------------------
5:
    IF fbElev.iCurrentFloor = 1 AND 
       fbElev.eState = E_ElevatorState.eIdle THEN
        bPassed := TRUE;
        bDone := TRUE;
    END_IF;

END_CASE;

// Call the function block every scan
//fbElev();

END_FUNCTION_BLOCK

// ---- POUs/FB_Dispatcher.TcPOU
FUNCTION_BLOCK FB_Dispatcher

// ============================================================================
// CONSTANTS
// ============================================================================
VAR CONSTANT
    cMAX_QUEUE_SIZE : INT := 50;
END_VAR

// ============================================================================
// INPUTS
// ============================================================================
VAR_INPUT
    // References to elevators (Composition pattern)
    refE1               : REFERENCE TO FB_Elevator;
    refE2               : REFERENCE TO FB_Elevator;
    
    // Traffic mode selection
    eTrafficMode        : E_TrafficMode := E_TrafficMode.eOffPeak;
    
    // System enable
    bEnable             : BOOL := TRUE;
END_VAR

// ============================================================================
// OUTPUTS
// ============================================================================
VAR_OUTPUT
    // Assignment tracking
    iAssignedToE1       : INT := 0;
    iAssignedToE2       : INT := 0;
    iUnassignedCalls    : INT := 0;
    
    // Performance metrics
    stMetrics           : ST_PerformanceMetrics;
END_VAR

// ============================================================================
// INTERNAL VARIABLES
// ============================================================================
VAR
    // Call queue
    _astCallQueue       : ARRAY[0..cMAX_QUEUE_SIZE] OF ST_FloorCall;
    _iQueueHead         : INT := 0;
    _iQueueTail         : INT := 0;
    _iQueueCount        : INT := 0;
    
    // Statistics
    _iTotalCalls        : DINT := 0;
    _fTotalWaitTime     : REAL := 0.0;
    _fMaxWaitTime       : REAL := 0.0;
    
    // Night mode
    _bNightModeActive   : BOOL := FALSE;
    _iActiveElevator    : INT := 1;
END_VAR

METHOD PUBLIC AddCall : BOOL
VAR_INPUT
    iFloor          : INT;
    eDirection      : E_Direction;
    bIsCarCall      : BOOL;
    iElevatorID     : INT;  // 0=hall call, 1=E1 car call, 2=E2 car call
END_VAR
IF _iQueueCount >= cMAX_QUEUE_SIZE THEN
    AddCall := FALSE;
    RETURN;
END_IF;

_astCallQueue[_iQueueTail].iFloor := iFloor;
_astCallQueue[_iQueueTail].eDirection := eDirection;
_astCallQueue[_iQueueTail].bIsCarCall := bIsCarCall;
_astCallQueue[_iQueueTail].tTimestamp := TIME();
_astCallQueue[_iQueueTail].iAssignedTo := 0;
_astCallQueue[_iQueueTail].bIsActive := TRUE;
_astCallQueue[_iQueueTail].tWaitTime := T#0S;

_iQueueTail := (_iQueueTail + 1) MOD (cMAX_QUEUE_SIZE + 1);
_iQueueCount := _iQueueCount + 1;
_iTotalCalls := _iTotalCalls + 1;

AddCall := TRUE;
END_METHOD

METHOD PRIVATE CalculateMetrics : BOOL
VAR
	fTotalDistance : REAL;
END_VAR
IF _iTotalCalls > 0 THEN
    stMetrics.fAvgResponseTime := _fTotalWaitTime / DINT_TO_REAL(_iTotalCalls);
ELSE
    stMetrics.fAvgResponseTime := 0.0;
END_IF;

stMetrics.fAvgWaitTime := stMetrics.fAvgResponseTime;
stMetrics.fMaxWaitTime := _fMaxWaitTime;

IF refE1.eState <> E_ElevatorState.eIdle AND 
   refE1.eState <> E_ElevatorState.eEmergencyStop THEN
    stMetrics.fUtilizationE1 := 85.0;
ELSE
    stMetrics.fUtilizationE1 := 15.0;
END_IF;

IF refE2.eState <> E_ElevatorState.eIdle AND 
   refE2.eState <> E_ElevatorState.eEmergencyStop THEN
    stMetrics.fUtilizationE2 := 85.0;
ELSE
    stMetrics.fUtilizationE2 := 15.0;
END_IF;

stMetrics.iCallsToday := _iTotalCalls;

fTotalDistance := refE1.fTravelDistance + refE2.fTravelDistance;
stMetrics.fEnergyEstimate := fTotalDistance * 0.15;

CalculateMetrics := TRUE;
END_METHOD

METHOD PUBLIC ClearAllCalls : BOOL
VAR
	i	: INT;
END_VAR
FOR i := 0 TO cMAX_QUEUE_SIZE DO
    _astCallQueue[i].bIsActive := FALSE;
END_FOR;

_iQueueCount := 0;
_iQueueHead := 0;
_iQueueTail := 0;

ClearAllCalls := TRUE;
END_METHOD

METHOD PUBLIC GetQueueStatus : AT_FloorCalls
VAR
	i : INT;
    j : INT := 0;
    aResult : AT_FloorCalls;
END_VAR
FOR i := 0 TO cMAX_QUEUE_SIZE DO
    IF _astCallQueue[i].bIsActive THEN
        aResult[j] := _astCallQueue[i];
        j := j + 1;
        IF j > cMAX_QUEUE_SIZE THEN
            EXIT;
        END_IF;
    END_IF;
END_FOR;

GetQueueStatus := aResult;
END_METHOD

METHOD ProcessQueue : BOOL
VAR
	i                   : INT;
    fScoreE1            : REAL;
    fScoreE2            : REAL;
    fDistanceE1         : REAL;
    fDistanceE2         : REAL;
    bE1CanServe         : BOOL;
    bE2CanServe         : BOOL;
    iE1Floor            : INT;
    iE2Floor            : INT;
    eE1Dir              : E_Direction;
    eE2Dir              : E_Direction;
    eE1State            : E_ElevatorState;
    eE2State            : E_ElevatorState;
END_VAR
IF NOT bEnable THEN
    ProcessQueue := FALSE;
    RETURN;
END_IF;


// 
iAssignedToE1 := 0;
iAssignedToE2 := 0;
iUnassignedCalls := 0;

// Get current elevator states
iE1Floor := refE1.iCurrentFloor;
iE2Floor := refE2.iCurrentFloor;
eE1Dir := refE1.eDirection;
eE2Dir := refE2.eDirection;
eE1State := refE1.eState;
eE2State := refE2.eState;

// Night mode handling
IF eTrafficMode = E_TrafficMode.eNightMode THEN
    IF NOT _bNightModeActive THEN
        _bNightModeActive := TRUE;
        IF _iActiveElevator = 1 THEN
            refE2.CallFloor(0);
        ELSE
            refE1.CallFloor(0);
        END_IF;
    END_IF;
ELSE
    _bNightModeActive := FALSE;
END_IF;

// Process each unassigned call
FOR i := 0 TO cMAX_QUEUE_SIZE DO
    IF _astCallQueue[i].bIsActive AND _astCallQueue[i].iAssignedTo = 0 THEN
        
        // Calculate distances
        fDistanceE1 := ABS(INT_TO_REAL(iE1Floor - _astCallQueue[i].iFloor));
        fDistanceE2 := ABS(INT_TO_REAL(iE2Floor - _astCallQueue[i].iFloor));
        
        // Direction compatibility
        bE1CanServe := (eE1Dir = E_Direction.eNone) OR 
                       (eE1Dir = _astCallQueue[i].eDirection) OR
                       _astCallQueue[i].bIsCarCall;
        bE2CanServe := (eE2Dir = E_Direction.eNone) OR 
                       (eE2Dir = _astCallQueue[i].eDirection) OR
                       _astCallQueue[i].bIsCarCall;
        
        // Base scores
        fScoreE1 := fDistanceE1;
        fScoreE2 := fDistanceE2;
        
        // Direction bonus
        IF bE1CanServe AND eE1Dir = _astCallQueue[i].eDirection THEN
            fScoreE1 := fScoreE1 * 0.6;
        END_IF;
        IF bE2CanServe AND eE2Dir = _astCallQueue[i].eDirection THEN
            fScoreE2 := fScoreE2 * 0.6;
        END_IF;
        
        // Traffic mode adjustments
        CASE eTrafficMode OF
            E_TrafficMode.eUpPeak:
                IF _astCallQueue[i].iFloor = 0 AND _astCallQueue[i].eDirection = E_Direction.eUp THEN
                    fScoreE1 := fScoreE1 * 0.7;
                END_IF;
                
            E_TrafficMode.eDownPeak:
                IF _astCallQueue[i].eDirection = E_Direction.eDown THEN
                    fScoreE2 := fScoreE2 * 0.7;
                END_IF;
                
            E_TrafficMode.eNightMode:
                IF _iActiveElevator = 1 THEN
                    fScoreE2 := 999.0;
                ELSE
                    fScoreE1 := 999.0;
                END_IF;
                
        END_CASE;
        
        // Availability check
        IF eE1State = E_ElevatorState.eEmergencyStop OR 
           eE1State = E_ElevatorState.eFireMode OR 
           eE1State = E_ElevatorState.eMaintenance THEN
            fScoreE1 := 999.0;
        END_IF;
        IF eE2State = E_ElevatorState.eEmergencyStop OR 
           eE2State = E_ElevatorState.eFireMode OR 
           eE2State = E_ElevatorState.eMaintenance THEN
            fScoreE2 := 999.0;
        END_IF;
        
        // Assign to best elevator
        IF fScoreE1 <= fScoreE2 THEN
            _astCallQueue[i].iAssignedTo := 1;
            refE1.CallFloor(_astCallQueue[i].iFloor);
            iAssignedToE1 := iAssignedToE1 + 1;
        ELSE
            _astCallQueue[i].iAssignedTo := 2;
            refE2.CallFloor(_astCallQueue[i].iFloor);
            iAssignedToE2 := iAssignedToE2 + 1;
        END_IF;
        
    END_IF;
END_FOR;

// Update completed calls and metrics
UpdateQueueStatus();
CalculateMetrics();

ProcessQueue := TRUE;
END_METHOD

METHOD PRIVATE UpdateQueueStatus : BOOL
VAR
	i : INT;
END_VAR
FOR i := 0 TO cMAX_QUEUE_SIZE DO
    IF _astCallQueue[i].bIsActive THEN
        
        // Update wait time
        _astCallQueue[i].tWaitTime := _astCallQueue[i].tWaitTime + TIME();
        
        // Check if call completed
        IF _astCallQueue[i].iAssignedTo = 1 THEN
            IF refE1.iCurrentFloor = _astCallQueue[i].iFloor AND 
               refE1.eState = E_ElevatorState.eDoorsOpen THEN
                _astCallQueue[i].bIsActive := FALSE;
                _iQueueCount := _iQueueCount - 1;
                
                _fTotalWaitTime := _fTotalWaitTime + TIME_TO_REAL(_astCallQueue[i].tWaitTime);
                IF TIME_TO_REAL(_astCallQueue[i].tWaitTime) > _fMaxWaitTime THEN
                    _fMaxWaitTime := TIME_TO_REAL(_astCallQueue[i].tWaitTime);
                END_IF;
            END_IF;
        ELSIF _astCallQueue[i].iAssignedTo = 2 THEN
            IF refE2.iCurrentFloor = _astCallQueue[i].iFloor AND 
               refE2.eState = E_ElevatorState.eDoorsOpen THEN
                _astCallQueue[i].bIsActive := FALSE;
                _iQueueCount := _iQueueCount - 1;
                
                _fTotalWaitTime := _fTotalWaitTime + TIME_TO_REAL(_astCallQueue[i].tWaitTime);
                IF TIME_TO_REAL(_astCallQueue[i].tWaitTime) > _fMaxWaitTime THEN
                    _fMaxWaitTime := TIME_TO_REAL(_astCallQueue[i].tWaitTime);
                END_IF;
            END_IF;
        END_IF;
        
    END_IF;
END_FOR;

UpdateQueueStatus := TRUE;
END_METHOD

END_FUNCTION_BLOCK

// ---- POUs/FB_Safety.TcPOU
FUNCTION_BLOCK FB_Safety

// ============================================================================
// CONSTANTS
// ============================================================================
VAR CONSTANT
    cMAX_ALARMS : INT := 99;
END_VAR

// ============================================================================
// INPUTS — Raw sensor signals
// ============================================================================
VAR_INPUT
    // Elevator references (to command them)
    refE1               : REFERENCE TO FB_Elevator;
    refE2               : REFERENCE TO FB_Elevator;
    
    // Door sensors (TRUE = obstruction detected)
    bE1DoorSensor       : BOOL := FALSE;
    bE2DoorSensor       : BOOL := FALSE;
    
    // Weight sensors (TRUE = overload)
    bE1WeightSensor     : BOOL := FALSE;
    bE2WeightSensor     : BOOL := FALSE;
    
    // Emergency stop buttons (TRUE = pressed)
    bE1EmergencyBtn     : BOOL := FALSE;
    bE2EmergencyBtn     : BOOL := FALSE;
    
    // Building safety
    bFireAlarm          : BOOL := FALSE;
    bFirefighterKey     : BOOL := FALSE;
    bPowerFault         : BOOL := FALSE;
    
    // Overspeed detectors
    bOverspeedE1        : BOOL := FALSE;
    bOverspeedE2        : BOOL := FALSE;
    
    // Door mechanism faults
    bDoorOpenFaultE1    : BOOL := FALSE;
    bDoorOpenFaultE2    : BOOL := FALSE;
END_VAR

// ============================================================================
// OUTPUTS — Safety decisions
// ============================================================================
VAR_OUTPUT
    bE1Enable           : BOOL := TRUE;
    bE2Enable           : BOOL := TRUE;
    bSystemAlarm        : BOOL := FALSE;
    sAlarmMessage       : STRING(120) := '';
    eAlarmSeverity      : E_AlarmSeverity := E_AlarmSeverity.eInfo;
    
    // Individual alarm flags
    bE1DoorObstruction  : BOOL := FALSE;
    bE2DoorObstruction  : BOOL := FALSE;
    bE1Overload         : BOOL := FALSE;
    bE2Overload         : BOOL := FALSE;
    bE1EmergencyActive  : BOOL := FALSE;
    bE2EmergencyActive  : BOOL := FALSE;
    bFireModeActive     : BOOL := FALSE;
END_VAR

// ============================================================================
// INTERNAL VARIABLES
// ============================================================================
VAR
    // Debounce timers
    _tonDoorObsE1       : TON;
    _tonDoorObsE2       : TON;
    _tonOverloadE1      : TON;
    _tonOverloadE2      : TON;
    _tonEmergencyE1     : TON;
    _tonEmergencyE2     : TON;
    _tonFireAlarm       : TON;
    _tonPowerFault      : TON;
    
    // Alarm history
    _astAlarmLog        : AT_AlarmLog;
    _iAlarmIndex        : INT := 0;
    _iNextEventID       : DINT := 1;
END_VAR

// ======================================================================
// DOOR OBSTRUCTION DETECTION
// ======================================================================
_tonDoorObsE1(IN := bE1DoorSensor, PT := T#200MS);
IF _tonDoorObsE1.Q THEN
    bE1DoorObstruction := TRUE;
    refE1.bDoorObstruction := TRUE;
    bSystemAlarm := TRUE;
    sAlarmMessage := 'E1 Door Obstruction Detected';
    eAlarmSeverity := E_AlarmSeverity.eWarning;
    AddAlarm(E_AlarmSeverity.eWarning, 1, 'E1 Door Obstruction', 'FB_Safety');
ELSE
    bE1DoorObstruction := FALSE;
    refE1.bDoorObstruction := FALSE;
END_IF;

_tonDoorObsE2(IN := bE2DoorSensor, PT := T#200MS);
IF _tonDoorObsE2.Q THEN
    bE2DoorObstruction := TRUE;
    refE2.bDoorObstruction := TRUE;
    bSystemAlarm := TRUE;
    sAlarmMessage := 'E2 Door Obstruction Detected';
    eAlarmSeverity := E_AlarmSeverity.eWarning;
    AddAlarm(E_AlarmSeverity.eWarning, 2, 'E2 Door Obstruction', 'FB_Safety');
ELSE
    bE2DoorObstruction := FALSE;
    refE2.bDoorObstruction := FALSE;
END_IF;

// ======================================================================
// OVERLOAD DETECTION
// ======================================================================
_tonOverloadE1(IN := bE1WeightSensor, PT := T#500MS);
IF _tonOverloadE1.Q THEN
    bE1Overload := TRUE;
    refE1.bOverload := TRUE;
    bE1Enable := FALSE;
    bSystemAlarm := TRUE;
    sAlarmMessage := 'E1 Overload - Service Suspended';
    eAlarmSeverity := E_AlarmSeverity.eCritical;
    AddAlarm(E_AlarmSeverity.eCritical, 1, 'E1 Overload Detected', 'FB_Safety');
ELSE
    bE1Overload := FALSE;
    refE1.bOverload := FALSE;
    bE1Enable := TRUE;
END_IF;

_tonOverloadE2(IN := bE2WeightSensor, PT := T#500MS);
IF _tonOverloadE2.Q THEN
    bE2Overload := TRUE;
    refE2.bOverload := TRUE;
    bE2Enable := FALSE;
    bSystemAlarm := TRUE;
    sAlarmMessage := 'E2 Overload - Service Suspended';
    eAlarmSeverity := E_AlarmSeverity.eCritical;
    AddAlarm(E_AlarmSeverity.eCritical, 2, 'E2 Overload Detected', 'FB_Safety');
ELSE
    bE2Overload := FALSE;
    refE2.bOverload := FALSE;
    bE2Enable := TRUE;
END_IF;

// ======================================================================
// EMERGENCY STOP
// ======================================================================
_tonEmergencyE1(IN := bE1EmergencyBtn, PT := T#100MS);
IF _tonEmergencyE1.Q THEN
    bE1EmergencyActive := TRUE;
    refE1.bEmergencyStop := TRUE;
    bSystemAlarm := TRUE;
    sAlarmMessage := 'E1 EMERGENCY STOP ACTIVATED';
    eAlarmSeverity := E_AlarmSeverity.eEmergency;
    AddAlarm(E_AlarmSeverity.eEmergency, 1, 'E1 Emergency Stop Button', 'FB_Safety');
END_IF;

_tonEmergencyE2(IN := bE2EmergencyBtn, PT := T#100MS);
IF _tonEmergencyE2.Q THEN
    bE2EmergencyActive := TRUE;
    refE2.bEmergencyStop := TRUE;
    bSystemAlarm := TRUE;
    sAlarmMessage := 'E2 EMERGENCY STOP ACTIVATED';
    eAlarmSeverity := E_AlarmSeverity.eEmergency;
    AddAlarm(E_AlarmSeverity.eEmergency, 2, 'E2 Emergency Stop Button', 'FB_Safety');
END_IF;

// Reset emergency when button released
IF NOT bE1EmergencyBtn AND bE1EmergencyActive THEN
    bE1EmergencyActive := FALSE;
    refE1.bEmergencyStop := FALSE;
    refE1.ResetEmergency();
END_IF;

IF NOT bE2EmergencyBtn AND bE2EmergencyActive THEN
    bE2EmergencyActive := FALSE;
    refE2.bEmergencyStop := FALSE;
    refE2.ResetEmergency();
END_IF;

// ======================================================================
// FIRE MODE
// ======================================================================
_tonFireAlarm(IN := bFireAlarm, PT := T#1S);
IF _tonFireAlarm.Q THEN
    bFireModeActive := TRUE;
    refE1.bFireMode := TRUE;
    refE2.bFireMode := TRUE;
    bSystemAlarm := TRUE;
    sAlarmMessage := 'FIRE MODE - ELEVATORS RETURNING TO GROUND';
    eAlarmSeverity := E_AlarmSeverity.eEmergency;
    AddAlarm(E_AlarmSeverity.eEmergency, 0, 'Building Fire Alarm Activated', 'FB_Safety');
END_IF;

// Firefighter override
IF bFirefighterKey THEN
    refE1.bFireMode := FALSE;
    refE2.bFireMode := FALSE;
    bFireModeActive := FALSE;
    sAlarmMessage := 'Firefighter Override Active';
    AddAlarm(E_AlarmSeverity.eWarning, 0, 'Firefighter Key Switch', 'FB_Safety');
END_IF;

// Reset fire mode when alarm clears
IF NOT bFireAlarm AND NOT bFirefighterKey AND bFireModeActive THEN
    bFireModeActive := FALSE;
    refE1.bFireMode := FALSE;
    refE2.bFireMode := FALSE;
    refE1.ResetFireMode();
    refE2.ResetFireMode();
END_IF;

// ======================================================================
// POWER FAULT
// ======================================================================
_tonPowerFault(IN := bPowerFault, PT := T#500MS);
IF _tonPowerFault.Q THEN
    bSystemAlarm := TRUE;
    sAlarmMessage := 'POWER FAULT DETECTED - BATTERY BACKUP ACTIVE';
    eAlarmSeverity := E_AlarmSeverity.eEmergency;
    AddAlarm(E_AlarmSeverity.eEmergency, 0, 'Power Supply Fault', 'FB_Safety');
END_IF;

// ======================================================================
// OVERSPEED PROTECTION
// ======================================================================
IF bOverspeedE1 THEN
    refE1.EmergencyStop();
    bSystemAlarm := TRUE;
    sAlarmMessage := 'E1 OVERSPEED - EMERGENCY BRAKE ACTIVATED';
    eAlarmSeverity := E_AlarmSeverity.eEmergency;
    AddAlarm(E_AlarmSeverity.eEmergency, 1, 'E1 Overspeed Detection', 'FB_Safety');
END_IF;

IF bOverspeedE2 THEN
    refE2.EmergencyStop();
    bSystemAlarm := TRUE;
    sAlarmMessage := 'E2 OVERSPEED - EMERGENCY BRAKE ACTIVATED';
    eAlarmSeverity := E_AlarmSeverity.eEmergency;
    AddAlarm(E_AlarmSeverity.eEmergency, 2, 'E2 Overspeed Detection', 'FB_Safety');
END_IF;

// ======================================================================
// DOOR FAULT DETECTION
// ======================================================================
IF bDoorOpenFaultE1 THEN
    bE1Enable := FALSE;
    bSystemAlarm := TRUE;
    sAlarmMessage := 'E1 Door Mechanism Fault';
    eAlarmSeverity := E_AlarmSeverity.eCritical;
    AddAlarm(E_AlarmSeverity.eCritical, 1, 'E1 Door Open/Close Fault', 'FB_Safety');
END_IF;

IF bDoorOpenFaultE2 THEN
    bE2Enable := FALSE;
    bSystemAlarm := TRUE;
    sAlarmMessage := 'E2 Door Mechanism Fault';
    eAlarmSeverity := E_AlarmSeverity.eCritical;
    AddAlarm(E_AlarmSeverity.eCritical, 2, 'E2 Door Open/Close Fault', 'FB_Safety');
END_IF;

METHOD PUBLIC AcknowledgeAlarm : BOOL
VAR_INPUT
    iEventID    : DINT;
    sOperator   : STRING(20);
END_VAR
VAR
    i : INT;
END_VAR
FOR i := 0 TO cMAX_ALARMS DO
    IF _astAlarmLog[i].iEventID = iEventID THEN
        _astAlarmLog[i].bAcknowledged := TRUE;
        _astAlarmLog[i].tAckTime := GetCurrentDateTime();
        _astAlarmLog[i].sAckBy := sOperator;
        AcknowledgeAlarm := TRUE;
        RETURN;
    END_IF;
END_FOR;

AcknowledgeAlarm := FALSE;
END_METHOD

METHOD PRIVATE AddAlarm : BOOL
VAR_INPUT
    eSeverity   : E_AlarmSeverity;
    iElevatorID : INT;
    sMessage    : STRING(120);
    sSource     : STRING(40);
END_VAR
_astAlarmLog[_iAlarmIndex].iEventID := _iNextEventID;
_iNextEventID := _iNextEventID + 1;

// Use current TIME for timestamp (simpler, no DT needed)
_astAlarmLog[_iAlarmIndex].tTimestamp := GetCurrentDateTime();
_astAlarmLog[_iAlarmIndex].eSeverity := eSeverity;
_astAlarmLog[_iAlarmIndex].iElevatorID := iElevatorID;
_astAlarmLog[_iAlarmIndex].sMessage := sMessage;
_astAlarmLog[_iAlarmIndex].sSource := sSource;
_astAlarmLog[_iAlarmIndex].bAcknowledged := FALSE;

_iAlarmIndex := (_iAlarmIndex + 1) MOD (cMAX_ALARMS + 1);

AddAlarm := TRUE;
END_METHOD

METHOD PUBLIC GetAlarmLog : AT_AlarmLog
VAR_INPUT
END_VAR
GetAlarmLog := _astAlarmLog;
END_METHOD

METHOD PRIVATE GetCurrentDateTime : DT
VAR
    ft : T_FILETIME;
    uliTime : ULINT;
END_VAR
uliTime := F_GetSystemTime();

ft.dwLowDateTime := TO_DWORD(uliTime AND 16#FFFFFFFF);
ft.dwHighDateTime := TO_DWORD(SHR(uliTime, 32));

GetCurrentDateTime := FILETIME_TO_DT(ft);
END_METHOD

METHOD PUBLIC ResetSystemAlarm : BOOL
VAR_INPUT
END_VAR
IF NOT bE1DoorSensor AND
   NOT bE2DoorSensor AND
   NOT bE1WeightSensor AND
   NOT bE2WeightSensor AND
   NOT bE1EmergencyBtn AND
   NOT bE2EmergencyBtn AND
   NOT bFireAlarm AND
   NOT bPowerFault AND
   NOT bOverspeedE1 AND
   NOT bOverspeedE2 AND
   NOT bDoorOpenFaultE1 AND
   NOT bDoorOpenFaultE2 THEN

    bSystemAlarm := FALSE;
    sAlarmMessage := '';
    eAlarmSeverity := E_AlarmSeverity.eInfo;

    ResetSystemAlarm := TRUE;
ELSE
    ResetSystemAlarm := FALSE;
END_IF
END_METHOD

END_FUNCTION_BLOCK
